{attribute 'qualified_only'}
VAR_GLOBAL CONSTANT
    stHmi : ST_HmiCommunicationConfig := (tWatchdogTimeout := T#2S);
    stGripper : ST_GripperCommunicationConfig := (tAdsTimeout := T#2S, tPollInterval := T#150MS);
    stCoaxVision : ST_VisionCommunicationConfig := (tResultTimeout := T#5S);
    stScrewVision : ST_VisionCommunicationConfig := (tResultTimeout := T#5S);
END_VAR

(* stored: Version 1.1.0.1, ProductVersion 3.1.4026.20
   GVL GVL_CommunicationConfig: Id {caf7f477-9eac-47d3-ac29-a9a22d445281} *)
